FUNCTION Or2 : BoolValue
VAR_INPUT
	value1 : BoolValue;
	value2 : BoolValue;
END_VAR
VAR
	p : POINTER TO BooleanExpression;
END_VAR

p := __NEW(BooleanExpression);

p^.Op2(
	operator := BooleanOperator.ORop,
	value1 := value1,
	value2 := value2
);

Or2 := p^;

END_FUNCTION

(* stored: Version 1.1.0.1
   POU Or2: Id {30a99ce2-ac44-4255-bac3-1519a0e516eb}, SpecialFunc None *)
